{attribute 'qualified_only'}
VAR_GLOBAL
END_VAR

(* stored: Version 1.1.0.1
   GVL GVL_1: Id {445610ce-1bd0-4a6e-9432-905d20da6b0b} *)
